PROGRAM Stn054_26_EmptyPuckStorageBreakStop2Grn
VAR
	{attribute 'TcLinkToOSO' := '
		.iPuckPresent :=  <0,1,1>TIIB[N56S00 (AL1332)]^N56S05 (AL2341)^TxPDO^input byte 1;
 		.iBufferFull  :=  <0,1,1>TIIB[N56S00 (AL1332)]^N56S05 (AL2341)^TxPDO^input byte 3;
		.oStopLower :=  <0,1,5>TIIB[N56S00 (AL1332)]^N56S02 (EX260)^RxPDO^output byte 1'}
	fbConvStop: FB_ConvStop;
END_VAR

//EmptyPuckStorageBreakStop2GRN  (7B)
//GRN Empty Puck Storage Break Stop 2 Puck Present
//GRN Empty Puck Storage Break Stop 2 DS Buffer


//  This code instantiates a component that is implimented as a common function block
//    Note that I/O is linked directly to I/O variables inside the named instance

gStn054_26_EmptyPuckStorageBreakStop2Grn.ConvRunning  := gConsumed_SafetyInterfaceConv.MtrRunning.Enc058Mtr03;

fbConvStop(
	pStn := ADR(gStn054),
	pCmp := ADR(gStn054_26_EmptyPuckStorageBreakStop2Grn),
	pUpstreamStop := 0,
	pStateTraceBuffer := ADR(gStn054_StateTraceBuffer),
	pStateTraceFifo := ADR(gStn054_StateTraceFifo),
	pStats := ADR(gStn054_02_Stats));

END_PROGRAM

(* stored: Version 1.1.0.1, ProductVersion 3.1.4024.6
   POU Stn054_26_EmptyPuckStorageBreakStop2Grn: Id {8995c99d-222f-477e-bbbe-e161dad9ae6b}, SpecialFunc None *)
